{attribute 'GeneratedUsingTerminal: ER8309-1022-0018'}
{attribute addProperty BoxType "ER8309-1022-0018"}
{attribute addProperty Id "StatusAT %I*Status_72C27E804"}
{attribute addProperty CRC "2006162193"}
{attribute addProperty Size "4"}
TYPE PWM_Status_77939B11 :
STRUCT
	{attribute addProperty Name "Status"}
	Status AT %I* : Status_72C27E80;
END_STRUCT
END_TYPE

(* stored: Version 1.2.0.0, ProductVersion 3.1.4024.9
   DUT PWM_Status_77939B11: Id {4f818cab-ac57-442c-8cb7-0304289040d8} *)
